PROGRAM Alarm_Display_ST
VAR
END_VAR

END_PROGRAM

(* stored: Version 1.1.0.1, ProductVersion 3.1.4024.0
   POU Alarm_Display_ST: Id {08e2e584-5ebd-4017-8838-0d3fbd977d4d}, SpecialFunc None *)
